(* CODESYS project WaterGAdoanddowhat.export

Project tree, tasks and I/O mapping:
  data type Do_WaterWhat
*)

// Do_WaterWhat
//{attribute 'qualified_only'}
//{attribute 'strict'}
TYPE Do_WaterWhat :
(
	Do_Filling,
	Do_Emptying
);
END_TYPE
